// SIMATIC STEP 7 (V5.x) project TEMA 5 EJERCICIO 48
// CPU: CPU313 C-2 DP(1)
// station: P_ADR_BUS
// station: Hardware
// station: Equipo SIMATIC 300
// program: Programa S7(1)

SYMBOL_TABLE
"FLANCOS"	DB 1	DB 1
"MANIOBRA"	DB 2	DB 2
"P MARCHA"	I 0.0	BOOL
"C FOTOELECTRICA"	I 0.1	BOOL
"P PARO"	I 0.2	BOOL
"CONTADOR"	MW 0	WORD
"Cycle Execution"	OB 1	OB 1
"LED PARO"	Q 0.0	BOOL
"LED MARCHA"	Q 0.1	BOOL
"C TRANSPORTADORA"	Q 0.2	BOOL
"PISTON EXPANDIDO"	Q 0.3	BOOL
"PISTON CONTRAIDO"	Q 0.4	BOOL
END_SYMBOL_TABLE

DATA_BLOCK "FLANCOS"	// DB 1
VERSION : 0.1
  STRUCT
   M0 : BOOL ;
   M1 : BOOL ;
   M2 : BOOL ;
   M3 : BOOL ;
   M4 : BOOL ;
   M5 : BOOL ;
   M6 : BOOL ;
   M7 : BOOL ;
   M10 : BOOL ;
   M11 : BOOL ;
   M12 : BOOL ;
   M13 : BOOL ;
   M14 : BOOL ;
   M15 : BOOL ;
   M16 : BOOL ;
   M17 : BOOL ;
   M20 : BOOL ;
   M21 : BOOL ;
   M22 : BOOL ;
   M23 : BOOL ;
   M24 : BOOL ;
   M25 : BOOL ;
   M26 : BOOL ;
   M27 : BOOL ;
  END_STRUCT ;	
BEGIN
END_DATA_BLOCK

DATA_BLOCK "MANIOBRA"	// DB 2
VERSION : 0.1
  STRUCT
   M0 : BOOL ;
   M1 : BOOL ;
   M2 : BOOL ;
   M3 : BOOL ;
   M4 : BOOL ;
   M5 : BOOL ;
   M6 : BOOL ;
   M7 : BOOL ;
  END_STRUCT ;	
BEGIN
END_DATA_BLOCK

ORGANIZATION_BLOCK "Cycle Execution"	// OB 1
TITLE = "Main Program Sweep (Cycle)"
//ENVASADOR DE MANZANAS
VERSION : 0.1
VAR_TEMP
  OB1_EV_CLASS : BYTE ;	//Bits 0-3 = 1 (Coming event), Bits 4-7 = 1 (Event class 1)
  OB1_SCAN_1 : BYTE ;	//1 (Cold restart scan 1 of OB 1), 3 (Scan 2-n of OB 1)
  OB1_PRIORITY : BYTE ;	//Priority of OB Execution
  OB1_OB_NUMBR : BYTE ;	//1 (Organization block 1, OB1)
  OB1_RESERVED_1 : BYTE ;	//Reserved for system
  OB1_RESERVED_2 : BYTE ;	//Reserved for system
  OB1_PREV_CYCLE : INT ;	//Cycle time of previous OB1 scan (milliseconds)
  OB1_MIN_CYCLE : INT ;	//Minimum cycle time of OB1 (milliseconds)
  OB1_MAX_CYCLE : INT ;	//Maximum cycle time of OB1 (milliseconds)
  OB1_DATE_TIME : DATE_AND_TIME ;	//Date and time OB1 started
END_VAR
BEGIN
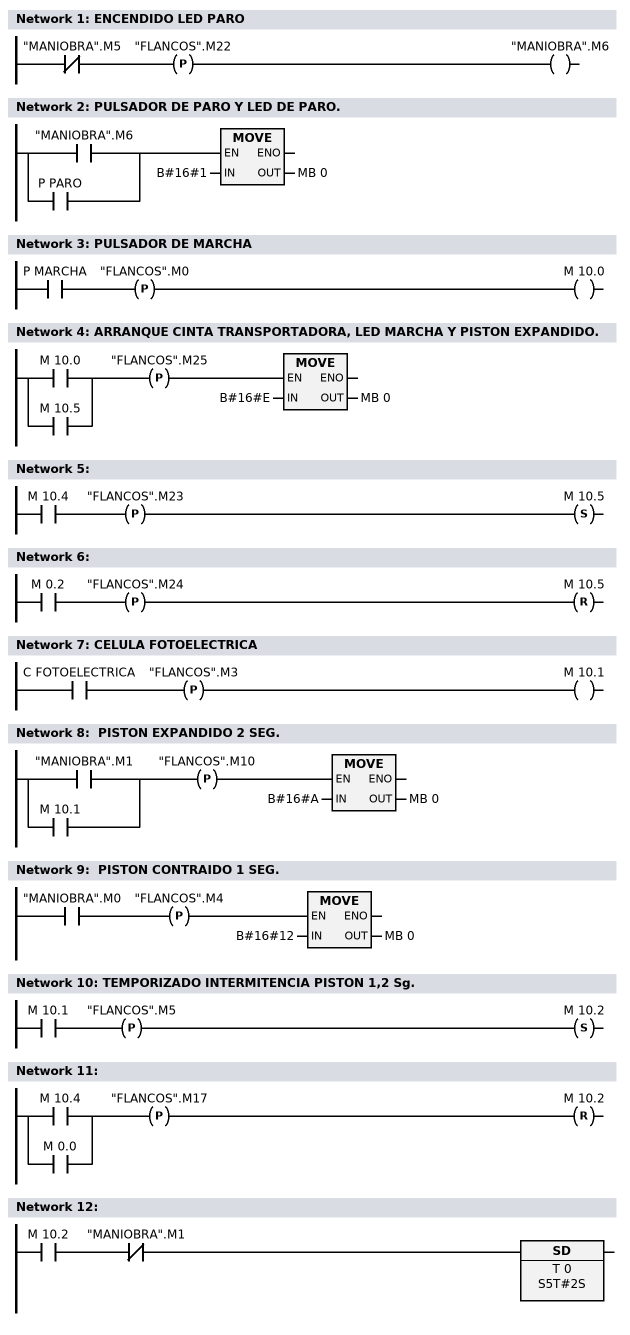
NETWORK
TITLE = ENCENDIDO LED PARO
      AN    "MANIOBRA".M5;
      FP    "FLANCOS".M22;
      =     "MANIOBRA".M6;
NETWORK
TITLE = PULSADOR DE PARO Y LED DE PARO.
      A(;
      O     "MANIOBRA".M6;
      O     "P PARO";
      );
      JNB   _001;
      L     B#16#1;
      T     MB 0;
_001: NOP   0;
NETWORK
TITLE = PULSADOR DE MARCHA
      A     "P MARCHA";
      FP    "FLANCOS".M0;
      =     M 10.0;
NETWORK
TITLE = ARRANQUE CINTA TRANSPORTADORA, LED MARCHA Y PISTON EXPANDIDO.
      A(;
      O     M 10.0;
      O     M 10.5;
      );
      FP    "FLANCOS".M25;
      JNB   _002;
      L     B#16#E;
      T     MB 0;
_002: NOP   0;
NETWORK
TITLE =
      A     M 10.4;
      FP    "FLANCOS".M23;
      S     M 10.5;
NETWORK
TITLE =
      A     M 0.2;
      FP    "FLANCOS".M24;
      R     M 10.5;
NETWORK
TITLE = CELULA FOTOELECTRICA
      A     "C FOTOELECTRICA";
      FP    "FLANCOS".M3;
      =     M 10.1;
NETWORK
TITLE =  PISTON EXPANDIDO 2 SEG.
      A(;
      O     "MANIOBRA".M1;
      O     M 10.1;
      );
      FP    "FLANCOS".M10;
      JNB   _003;
      L     B#16#A;
      T     MB 0;
_003: NOP   0;
NETWORK
TITLE =  PISTON CONTRAIDO 1 SEG.
      A     "MANIOBRA".M0;
      FP    "FLANCOS".M4;
      JNB   _004;
      L     B#16#12;
      T     MB 0;
_004: NOP   0;
NETWORK
TITLE = TEMPORIZADO INTERMITENCIA PISTON 1,2 Sg.
      A     M 10.1;
      FP    "FLANCOS".M5;
      S     M 10.2;
NETWORK
TITLE =
      A(;
      O     M 10.4;
      O     M 0.0;
      );
      FP    "FLANCOS".M17;
      R     M 10.2;
NETWORK
TITLE =  
      A     M 10.2;
      AN    "MANIOBRA".M1;
      L     S5T#2S;
      SD    T 0;
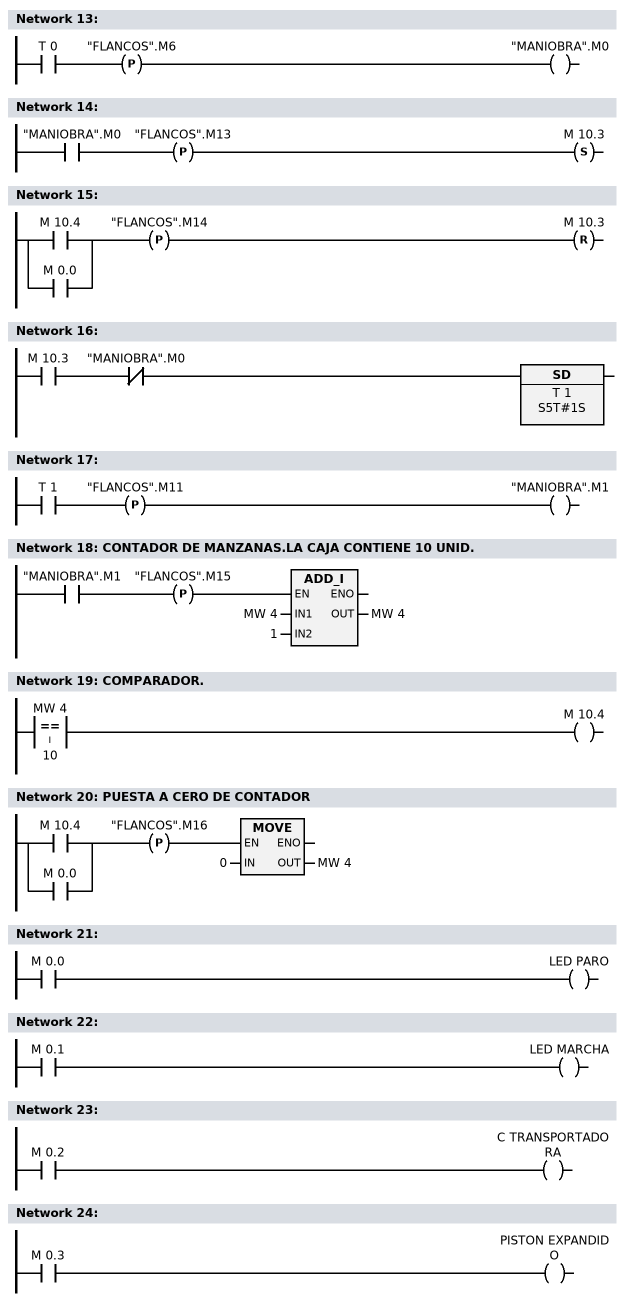
NETWORK
TITLE =
      A     T 0;
      FP    "FLANCOS".M6;
      =     "MANIOBRA".M0;
NETWORK
TITLE =
      A     "MANIOBRA".M0;
      FP    "FLANCOS".M13;
      S     M 10.3;
NETWORK
TITLE =
      A(;
      O     M 10.4;
      O     M 0.0;
      );
      FP    "FLANCOS".M14;
      R     M 10.3;
NETWORK
TITLE =
      A     M 10.3;
      AN    "MANIOBRA".M0;
      L     S5T#1S;
      SD    T 1;
NETWORK
TITLE =
      A     T 1;
      FP    "FLANCOS".M11;
      =     "MANIOBRA".M1;
NETWORK
TITLE = CONTADOR DE MANZANAS.LA CAJA CONTIENE 10 UNID.
      A     "MANIOBRA".M1;
      FP    "FLANCOS".M15;
      JNB   _005;
      L     MW 4;
      L     1;
      +I;
      T     MW 4;
_005: NOP   0;
NETWORK
TITLE = COMPARADOR.
//PONE A CERO CONTADOR ,DESACTIVA INTERMITENCIA PISTON Y ARRANCA CINTA 
//TRANSPORTADORA.
      L     MW 4;
      L     10;
      ==I;
      =     M 10.4;
NETWORK
TITLE = PUESTA A CERO DE CONTADOR
      A(;
      O     M 10.4;
      O     M 0.0;
      );
      FP    "FLANCOS".M16;
      JNB   _006;
      L     0;
      T     MW 4;
_006: NOP   0;
NETWORK
TITLE =
      A     M 0.0;
      =     "LED PARO";
NETWORK
TITLE =
      A     M 0.1;
      =     "LED MARCHA";
NETWORK
TITLE =
      A     M 0.2;
      =     "C TRANSPORTADORA";
NETWORK
TITLE =
      A     M 0.3;
      =     "PISTON EXPANDIDO";
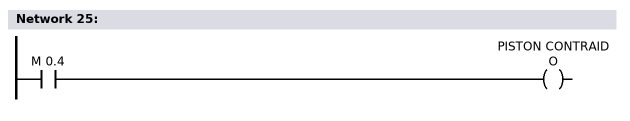
NETWORK
TITLE =
      A     M 0.4;
      =     "PISTON CONTRAIDO";
END_ORGANIZATION_BLOCK
